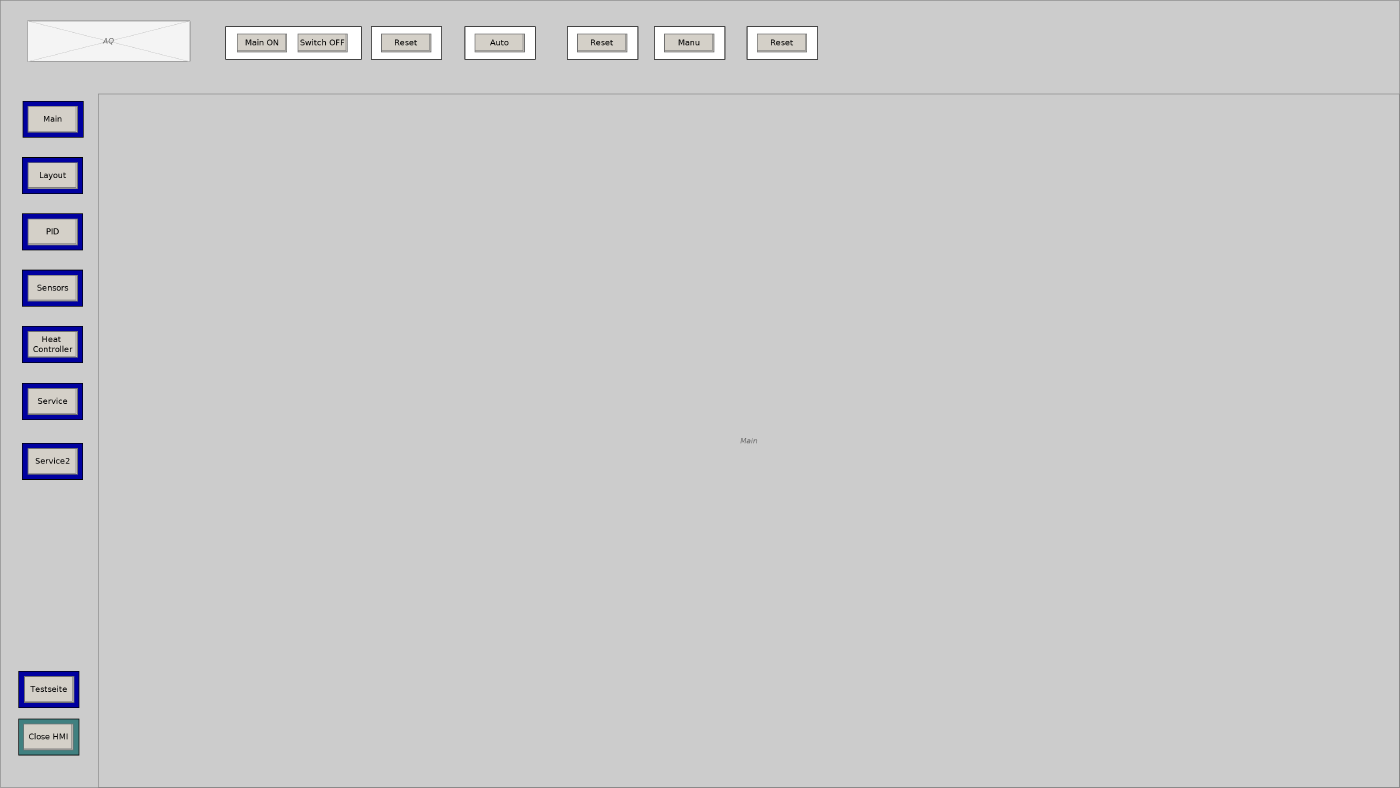
VISUALIZATION FRAME  // 1914x1078
    Frame (134,128 1780x950)
        shows Main()
        shows Heatreg()
        shows Sensors()
        shows Service()
        shows Layout()
        shows PID()
        shows Testseite1()
        shows PID_alt()
    Rectangle (30,215 83x50)
    Rectangle (31,138 83x50)
    Rectangle (30,292 83x50)
    Rectangle (30,369 83x50)
    Rectangle (30,446 83x50)
    Rectangle (30,524 83x50)
    Button (38,145 68x36), "Main"
        OnMouseDown: FrameSelectionChange Selection=SelectedFrame=19e204b9-edb1-49a7-b794-f10e0e8216a7, GlobSel=AssignType=Directly, SelType=Locally
    Rectangle (308,36 186x45), colour toggle: GVL.Mainswitch_OK
    Rectangle (507,36 97x45), colour toggle: GVL.ERROR_Mainswitch
    Rectangle (635,36 97x45), colour toggle: GVL.Control_Auto_active
    Rectangle (775,36 97x45), colour toggle: GVL.Reset_auto
    Rectangle (894,36 97x45), colour toggle: GVL.Control_Manu_active
    Rectangle (1021,36 97x45), colour toggle: GVL.Reset_man
    Button (324,46 68x25), "Main ON"
        tap GVL.Start_Mainswitch
    Button (407,46 68x25), "Switch OFF"
        tap GVL.Switch_OFF_Mainswitch
    Button (521,46 68x25), "Reset"
        tap GVL.RESET_ERROR_Mainswitch
    Button (649,46 68x25), "Auto"
        tap GVL.Control_Auto
    Button (789,46 68x25), "Reset"
        tap GVL.Reset_auto
    Button (908,46 68x25), "Manu"
        tap GVL.Control_Manu
    Button (1035,46 68x25), "Reset"
        tap GVL.Reset_man
    Image (37,28 223x56), image: AQ
    Button (38,222 68x36), "Layout"
        OnMouseDown: FrameSelectionChange Selection=SelectedFrame=19e204b9-edb1-49a7-b794-f10e0e8216a7, Selection=4, GlobSel=AssignType=Directly, SelType=Locally
    Button (38,299 68x36), "PID"
        OnMouseDown: FrameSelectionChange Selection=SelectedFrame=19e204b9-edb1-49a7-b794-f10e0e8216a7, Selection=5, GlobSel=AssignType=Directly, SelType=Locally
    Button (38,376 68x36), "Sensors"
        OnMouseDown: FrameSelectionChange Selection=SelectedFrame=19e204b9-edb1-49a7-b794-f10e0e8216a7, Selection=2, GlobSel=AssignType=Directly, SelType=Locally
    Button (38,453 68x36), "Heat Controller"
        OnMouseDown: FrameSelectionChange Selection=SelectedFrame=19e204b9-edb1-49a7-b794-f10e0e8216a7, Selection=1, GlobSel=AssignType=Directly, SelType=Locally
    Button (38,531 68x36), "Service"
        OnMouseDown: FrameSelectionChange Selection=SelectedFrame=19e204b9-edb1-49a7-b794-f10e0e8216a7, Selection=3, GlobSel=AssignType=Directly, SelType=Locally
    Rectangle (25,983 83x50)
    Button (32,990 68x36), "Close HMI"
        OnMouseDown: FrameSelectionChange Selection=SelectedFrame=19e204b9-edb1-49a7-b794-f10e0e8216a7, Selection=4, GlobSel=AssignType=Directly, SelType=Locally
        OnMouseDown: ExecuteCommand 
        OnMouseDown: CloseDialog Dialog=FileOpenSave, Result=OK, NumpadKeypadSet=True
        OnMouseDown: OpenDialog OpenModal=True, OpenCentered=True
        OnMouseDown: ExecuteCommand 
        OnMouseDown: execute {  }
        OnMouseDown: execute {  }
        OnMouseDown: ExecuteCommand ExecuteCommand=ExecuteCommand=[Command=ExecuteClientProgram, Value='TASKKILL /IM', Value2='Tc3PlcHMI.exe']
    Rectangle (25,918 83x50)
    Button (33,925 68x36), "Testseite"
        OnMouseDown: FrameSelectionChange Selection=SelectedFrame=19e204b9-edb1-49a7-b794-f10e0e8216a7, Selection=6, GlobSel=AssignType=Directly, SelType=Locally
    Rectangle (30,606 83x50)
    Button (38,613 68x36), "Service2"
        OnMouseDown: FrameSelectionChange Selection=SelectedFrame=19e204b9-edb1-49a7-b794-f10e0e8216a7, Selection=7, GlobSel=AssignType=Directly, SelType=Locally
END_VISUALIZATION

(* stored: Version 1.1.0.1, ProductVersion 3.1.4024.3
   Visu FRAME: Id {e4a26c6b-2bbb-4630-ad23-8c499fc78d66} *)
